// Mitsubishi GX Works2 project: 20250407_최종프로젝트_PLC_완성   PLC: Q03UDE

// global labels: Global1
VAR_GLOBAL
  압착1전솔 AT Y30 : BOOL;
  압착2전솔 AT Y31 : BOOL;
  배출전솔 AT Y32 : BOOL;
  회전전솔 AT Y34 : BOOL;
  회전후솔 AT Y35 : BOOL;
  스탑전솔 AT Y36 : BOOL;
  스탑후솔 AT Y37 : BOOL;
  서보전솔 AT Y38 : BOOL;
  서보후솔 AT Y39 : BOOL;
  컨베이어1 AT Y20 : BOOL;
  컨베이어2 AT Y21 : BOOL;
  컨베이어3 AT Y22 : BOOL;
  컨베이어4 AT Y23 : BOOL;
  스톱전센서 AT X1 : BOOL;
  스톱후센서 AT X0 : BOOL;
  스톱감지광센서 AT X2 : BOOL;
  두봇감지광센서1 AT X3 : BOOL;
  압착하강센서1 AT X5 : BOOL;
  회전상승센서 AT X7 : BOOL;
  회전하강센서 AT X8 : BOOL;
  배출감지광센서 AT X9 : BOOL;
  포장감지광센서1 AT X0A : BOOL;
  압착상승센서2 AT X0B : BOOL;
  압착하강센서2 AT X0C : BOOL;
  서보적재전센서 AT X0D : BOOL;
  서보적재후센서 AT X0E : BOOL;
  압착상승센서1 AT X6 : BOOL;
  포장감지광센서2 AT X10 : BOOL;
  회전감지광센서 AT X11 : BOOL;
  배출후센서 AT X13 : BOOL;
  배출전센서 AT X12 : BOOL;
  압착감지광센서 AT X14 : BOOL;
  두봇1빨강 AT Y2C : BOOL;
  두봇1하늘 AT Y2D : BOOL;
  두봇1노랑 AT Y2E : BOOL;
  두봇2동작1 AT Y2B : BOOL;
  축1서보기동번호 AT U4\G1500 : DINT;
  축1서보조그스피드값 AT U4\G1518 : DINT;
  축1서보현재위치 AT U4\G800 : DINT;
  축1서보이송속도 AT U4\G804 : DINT;
  축1서보원점복귀완료 AT U4\G817.4 : BOOL;
  QD75레디 AT X40 : BOOL;
  축1서보비지 AT X4C : BOOL;
  축1서보완료 AT X54 : BOOL;
  PLC레디 AT Y40 : BOOL;
  축1서보정지 AT Y44 : BOOL;
  축1서보조그정기동 AT Y48 : BOOL;
  축1서보조그역기동 AT Y49 : BOOL;
  축1서보기동 AT Y50 : BOOL;
  축2서보기동번호 AT U4\G1600 : DINT;
  축2서보조그스피드값 AT U4\G1618 : DINT;
  축2서보현재위치 AT U4\G900 : DINT;
  축2서보이송속도 AT U4\G904 : DINT;
  축2서보원점복귀완료 AT U4\G917.4 : BOOL;
  축2서보비지 AT X4B : BOOL;
  축2서보완료 AT X55 : BOOL;
  축2서보정지 AT Y45 : BOOL;
  축2서보조그정기동 AT Y4A : BOOL;
  축2서보조그역기동 AT Y4B : BOOL;
  축2서보기동 AT Y51 : BOOL;
  축1서보현재위치표시 AT D0 : DINT;
  축2서보현재위치표시 AT D10 : DINT;
  축1서보조그속도 AT D20 : DINT;
  축2서보조그속도 AT D30 : DINT;
  H1조그상 AT M0 : BOOL;
  H1조그하 AT M1 : BOOL;
  H2조그상 AT M2 : BOOL;
  H2조그하 AT M3 : BOOL;
  H1원점복귀버튼 AT M4 : BOOL;
  축1에러번호 AT U4\G806 : INT;
  축2에러번호 AT U4\G906 : INT;
  축1경고번호 AT U4\G807 : INT;
  축2경고번호 AT U4\G907 : INT;
  H시작버튼 AT M5 : BOOL;
  H일시정지버튼 AT M6 : BOOL;
  H비상정지버튼 AT M7 : BOOL;
  녹색램프 AT Y24 : BOOL;
  황색램프 AT Y25 : BOOL;
  적색램프 AT Y26 : BOOL;
  H축1원점복귀버튼 AT M8 : BOOL;
  H축2원점복귀버튼 AT M9 : BOOL;
  H롬저장 AT M200 : BOOL;
  서보롬쓰기 AT U4\G1900 : INT;
  H축1위치1입력 AT M300 : BOOL;
  H축1위치2입력 AT M301 : BOOL;
  H축1위치3입력 AT M302 : BOOL;
  H축2위치1입력 AT M310 : BOOL;
  H축2위치2입력 AT M311 : BOOL;
  H축2위치3입력 AT M312 : BOOL;
  H축2위치4입력 AT M313 : BOOL;
  H축2위치5입력 AT M314 : BOOL;
  H축2위치6입력 AT M315 : BOOL;
  H서보전진버튼 AT M10 : BOOL;
  H서보후진버튼 AT M11 : BOOL;
  H축1경고번호 AT D100 : INT;
  H축1에러번호 AT D101 : INT;
  H축2경고번호 AT D200 : INT;
  H축2에러번호 AT D201 : INT;
  H축1에러리셋 AT M400 : BOOL;
  H축2에러리셋 AT M401 : BOOL;
  축1에러리셋 AT U4\G1502 : INT;
  축2에러리셋 AT U4\G1602 : INT;
  송신채널 AT D1000 : INT;
  송신데이터수 AT D1002 : INT;
  송신데이터 AT D1010 : INT;
  수신채널 AT D1100 : INT;
  수신데이터수 AT D1103 : INT;
  수신버퍼 AT D1110 : INT;
  데이터체크 AT D1200 : INT;
  수신데이터확인 AT X6A : BOOL;
  송신정상 AT M1000 : BOOL;
  수신정상 AT M1100 : BOOL;
  두봇1완료 AT X18 : BOOL;
  두봇2완료 AT X19 : BOOL;
  H실린더스톱전진 AT M100 : BOOL;
  H실린더배출전진 AT M102 : BOOL;
  H실린더서보전진 AT M103 : BOOL;
  H실린더서보후진 AT M104 : BOOL;
  H실린더회전전진 AT M105 : BOOL;
  H실린더회전후진 AT M106 : BOOL;
  H실린더스톱후진 AT M101 : BOOL;
  H실린더압착전진1 AT M107 : BOOL;
  H실린더압착전진2 AT M108 : BOOL;
  H모터컨베이어1 AT M109 : BOOL;
  H모터컨베이어2 AT M110 : BOOL;
  H모터컨베이어3 AT M111 : BOOL;
  H모터컨베이어4 AT M112 : BOOL;
  S공정1_CT AT D3000 : INT;
  S공정2_CT AT D3002 : INT;
  S공정3_CT AT D3004 : INT;
  S공정4_CT AT D3006 : INT;
  축1서보조그속도표시 AT D40 : DINT;
  축2서보조그속도표시 AT D50 : DINT;
  S양품갯수 AT D3008 : INT;
  S불량갯수 AT D3010 : INT;
  S적재갯수 AT D3012 : INT;
  S고배율갯수 AT D3014 : INT;
  S중배율갯수 AT D3015 : INT;
  S저배율갯수 AT D3016 : INT;
  S고배율 AT D3017 : INT;
  S중배율 AT D3018 : INT;
  S저배율 AT D3019 : INT;
  두봇2동작중 AT M17 : BOOL;
  두봇1동작중 AT M16 : BOOL;
  녹색램프버튼 AT M30 : BOOL;
  황색램프버튼 AT M31 : BOOL;
  적색램프버튼 AT M32 : BOOL;
END_VAR

PROGRAM MAIN
VAR
  공정시작 : BOOL;
  축2기동 : BOOL;
  축1기동 : BOOL;
  공정종료 : BOOL;
  스톱후진 : BOOL;
  컨베이어1구동 : BOOL;
  컨베이어1정지 : BOOL;
  스톱전진 : BOOL;
  T스톱지연 : TIMER;
  서보준비완료 : BOOL;
  두봇앞정지 : BOOL;
  컨베이어1정지2 : BOOL;
  T두봇지연 : TIMER;
  압착앞이동 : BOOL;
  압착압이동 : BOOL;
  압착1전진 : BOOL;
  압착1후진 : BOOL;
  컨베이어1정지3 : BOOL;
  압착전진 : BOOL;
  압착후진 : BOOL;
  컨베이어1종료 : BOOL;
  T컨베이어1지연 : TIMER;
  컨베이어2구동 : BOOL;
  공정1종료 : BOOL;
  컨베이어1정지4 : BOOL;
  컨베이어4구동 : BOOL;
  T불량품감지 : TIMER;
  컨베이어3구동 : BOOL;
  컨베이어2정지1 : BOOL;
  비전감지 : BOOL;
  T비전감지지연 : TIMER;
  양품판별 : BOOL;
  불량판별 : BOOL;
  T두봇지연2 : TIMER;
  T포장1지연 : TIMER;
  T두봇지연3 : TIMER;
  T압착지연 : TIMER;
  압착2전진 : BOOL;
  압착2후진 : BOOL;
  회전전진 : BOOL;
  서보위치1이동 : BOOL;
  서보전진 : BOOL;
  T회전지연 : TIMER;
  T비상정지초기화 : TIMER;
  포장대기 : BOOL;
  포장대기2 : BOOL;
  축1위치1이동 : BOOL;
  축2위치1이동 : BOOL;
  T서보전진지연 : TIMER;
  서보후진 : BOOL;
  T서보후진지연 : TIMER;
  축2위치2이동 : BOOL;
  회전후진 : BOOL;
  축2위치3이동 : BOOL;
  축1위치2이동 : BOOL;
  축2위치4이동 : BOOL;
  T서보전진지연2 : TIMER;
  축1위치1이동2 : BOOL;
  축2위치1이동2 : BOOL;
  축2위치3이동2 : BOOL;
  회전대기 : BOOL;
  축1원점복귀 : BOOL;
  축2원점복귀 : BOOL;
  양품개수 : INT;
  연속종료 : BOOL;
  서보적재후진 : BOOL;
  롬쓰기 : BOOL;
  H롬쓰기 : BOOL;
  축1조그스피드값 : DINT;
  축2조그스피드값 : DINT;
  T압착정지지연 : TIMER;
  T압착정지지연2 : TIMER;
  공정중 : BOOL;
  적재완료대기 : BOOL;
  스톱후진2 : BOOL;
  T회전후진지연 : TIMER;
  시작 : BOOL;
  종료복귀 : BOOL;
  축1복귀1이동 : BOOL;
  복귀종료 : BOOL;
  축2복귀1이동 : BOOL;
  축1복귀2이동 : BOOL;
  종료 : BOOL;
  T불량판별지연 : TIMER;
  배출전진 : BOOL;
  배출후진 : BOOL;
  불량종료 : BOOL;
  양품종료 : BOOL;
  컨종료 : BOOL;
  T컨종료지연 : TIMER;
  두봇사양구별 : BOOL;
  두봇1완료신호 : BOOL;
  T포장대기지연 : TIMER;
  두봇포장완료 : BOOL;
  T컨베이어4지연 : TIMER;
  테스트 : BOOL;
  공정1그래프 : BOOL;
  공정2그래프 : BOOL;
  공정3그래프 : BOOL;
  공정4그래프 : BOOL;
  공정1CT : INT;
  공정2CT : INT;
  공정3CT : INT;
  공정4CT : INT;
  불량개수 : INT;
  적재완료 : BOOL;
  스톱후진3 : BOOL;
  두봇2동작 : BOOL;
  축1일시정지요구 : BOOL;
  축2일시정지요구 : BOOL;
  축2비상정지요구 : BOOL;
  축1비상정지요구 : BOOL;
  비상정지요구 : BOOL;
  일시정지요구 : BOOL;
  T축2일시정지기동 : TIMER;
  일시정지풀림 : BOOL;
END_VAR
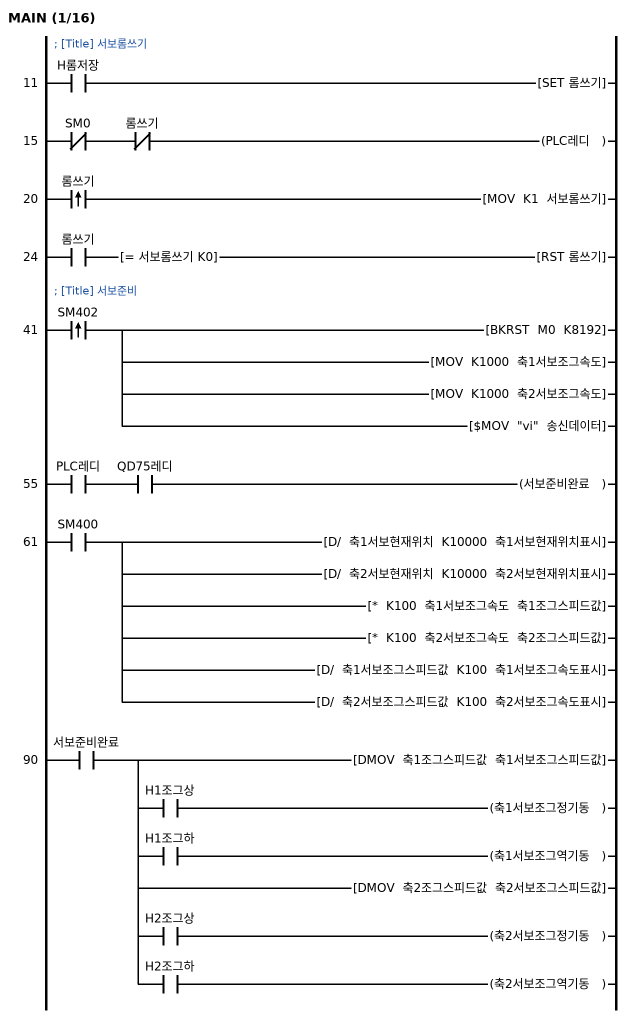
; [Title] 서보롬쓰기
11    LD      H롬저장
      SET     롬쓰기
15    LDI     SM0
      ANI     롬쓰기
      OUT     PLC레디
20    LDP     롬쓰기
      MOV     K1 서보롬쓰기
24    LD      롬쓰기
      AND=    서보롬쓰기 K0
      RST     롬쓰기
; [Title] 서보준비
41    LDP     SM402
      BKRST   M0 K8192
      MOV     K1000 축1서보조그속도
      MOV     K1000 축2서보조그속도
      $MOV    "vi" 송신데이터
55    LD      PLC레디
      AND     QD75레디
      OUT     서보준비완료
61    LD      SM400
      D/      축1서보현재위치 K10000 축1서보현재위치표시
      D/      축2서보현재위치 K10000 축2서보현재위치표시
      *       K100 축1서보조그속도 축1조그스피드값
      *       K100 축2서보조그속도 축2조그스피드값
      D/      축1서보조그스피드값 K100 축1서보조그속도표시
      D/      축2서보조그스피드값 K100 축2서보조그속도표시
90    LD      서보준비완료
      DMOV    축1조그스피드값 축1서보조그스피드값
      MPS
      AND     H1조그상
      OUT     축1서보조그정기동
      MRD
      AND     H1조그하
      OUT     축1서보조그역기동
      MPP
      DMOV    축2조그스피드값 축2서보조그스피드값
      MPS
      AND     H2조그상
      OUT     축2서보조그정기동
      MPP
      AND     H2조그하
      OUT     축2서보조그역기동
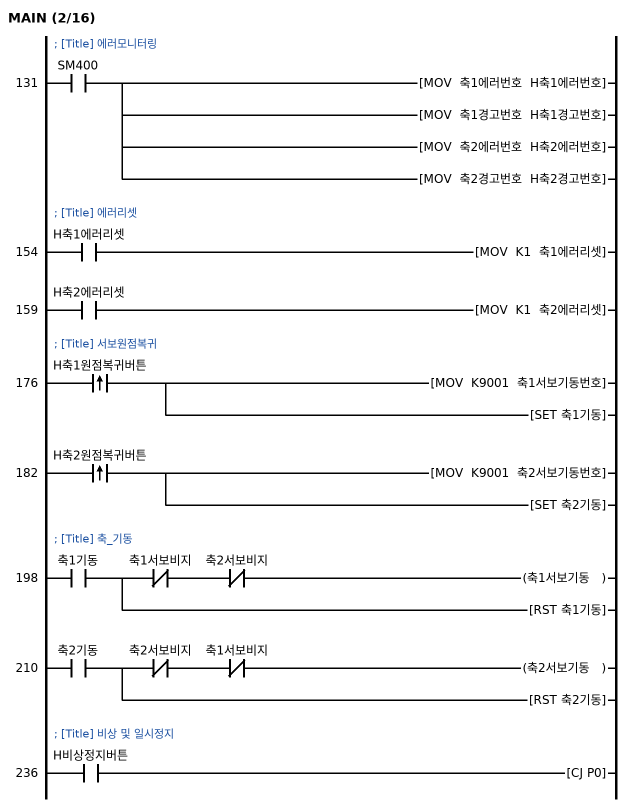
; [Title] 에러모니터링
131   LD      SM400
      MOV     축1에러번호 H축1에러번호
      MOV     축1경고번호 H축1경고번호
      MOV     축2에러번호 H축2에러번호
      MOV     축2경고번호 H축2경고번호
; [Title] 에러리셋
154   LD      H축1에러리셋
      MOV     K1 축1에러리셋
159   LD      H축2에러리셋
      MOV     K1 축2에러리셋
; [Title] 서보원점복귀
176   LDP     H축1원점복귀버튼
      MOV     K9001 축1서보기동번호
      SET     축1기동
182   LDP     H축2원점복귀버튼
      MOV     K9001 축2서보기동번호
      SET     축2기동
; [Title] 축_기동
198   LD      축1기동
      MPS
      ANI     축1서보비지
      ANI     축2서보비지
      OUT     축1서보기동
      MPP
      RST     축1기동
210   LD      축2기동
      MPS
      ANI     축2서보비지
      ANI     축1서보비지
      OUT     축2서보기동
      MPP
      RST     축2기동
; [Title] 비상 및 일시정지
236   LD      H비상정지버튼
      CJ      P0
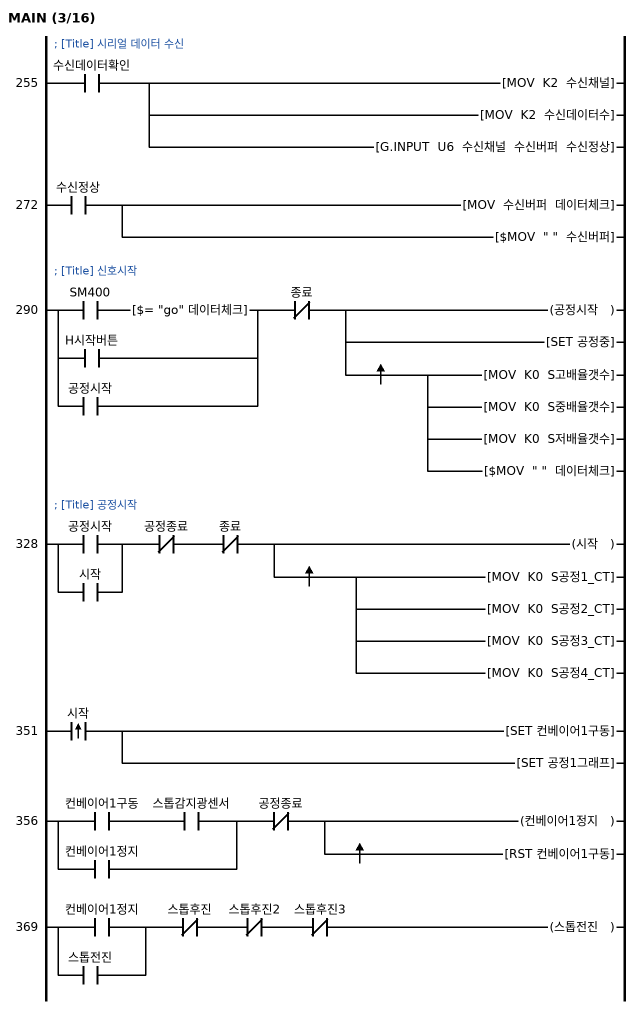
; [Title] 시리얼 데이터 수신
255   LD      수신데이터확인
      MOV     K2 수신채널
      MOV     K2 수신데이터수
      G.INPUT U6 수신채널 수신버퍼 수신정상
272   LD      수신정상
      MOV     수신버퍼 데이터체크
      $MOV    "" 수신버퍼
; [Title] 신호시작
290   LD      SM400
      AND$=   "go" 데이터체크
      OR      H시작버튼
      OR      공정시작
      ANI     종료
      OUT     공정시작
      SET     공정중
      MEP
      MOV     K0 S고배율갯수
      MOV     K0 S중배율갯수
      MOV     K0 S저배율갯수
      $MOV    "" 데이터체크
; [Title] 공정시작
328   LD      공정시작
      OR      시작
      ANI     공정종료
      ANI     종료
      OUT     시작
      MEP
      MOV     K0 S공정1_CT
      MOV     K0 S공정2_CT
      MOV     K0 S공정3_CT
      MOV     K0 S공정4_CT
351   LDP     시작
      SET     컨베이어1구동
      SET     공정1그래프
356   LD      컨베이어1구동
      AND     스톱감지광센서
      OR      컨베이어1정지
      ANI     공정종료
      OUT     컨베이어1정지
      MEP
      RST     컨베이어1구동
369   LD      컨베이어1정지
      OR      스톱전진
      ANI     스톱후진
      ANI     스톱후진2
      ANI     스톱후진3
      OUT     스톱전진
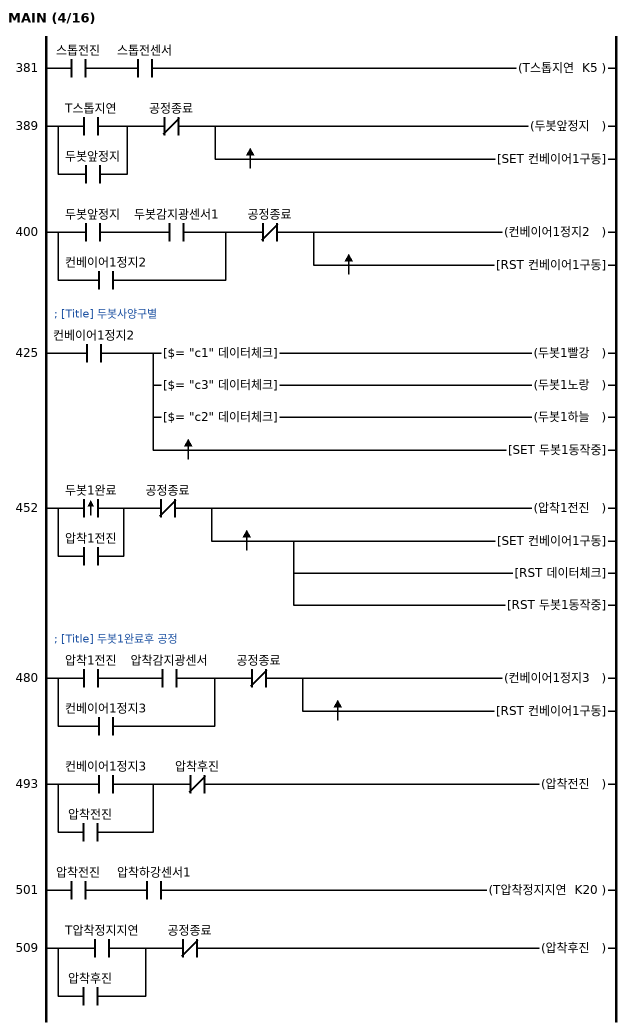
381   LD      스톱전진
      AND     스톱전센서
      OUT     T스톱지연 K5
389   LD      T스톱지연
      OR      두봇앞정지
      ANI     공정종료
      OUT     두봇앞정지
      MEP
      SET     컨베이어1구동
400   LD      두봇앞정지
      AND     두봇감지광센서1
      OR      컨베이어1정지2
      ANI     공정종료
      OUT     컨베이어1정지2
      MEP
      RST     컨베이어1구동
; [Title] 두봇사양구별
425   LD      컨베이어1정지2
      MPS
      AND$=   "c1" 데이터체크
      OUT     두봇1빨강
      MRD
      AND$=   "c3" 데이터체크
      OUT     두봇1노랑
      MRD
      AND$=   "c2" 데이터체크
      OUT     두봇1하늘
      MPP
      MEP
      SET     두봇1동작중
452   LDP     두봇1완료
      OR      압착1전진
      ANI     공정종료
      OUT     압착1전진
      MEP
      SET     컨베이어1구동
      RST     데이터체크
      RST     두봇1동작중
; [Title] 두봇1완료후 공정
480   LD      압착1전진
      AND     압착감지광센서
      OR      컨베이어1정지3
      ANI     공정종료
      OUT     컨베이어1정지3
      MEP
      RST     컨베이어1구동
493   LD      컨베이어1정지3
      OR      압착전진
      ANI     압착후진
      OUT     압착전진
501   LD      압착전진
      AND     압착하강센서1
      OUT     T압착정지지연 K20
509   LD      T압착정지지연
      OR      압착후진
      ANI     공정종료
      OUT     압착후진
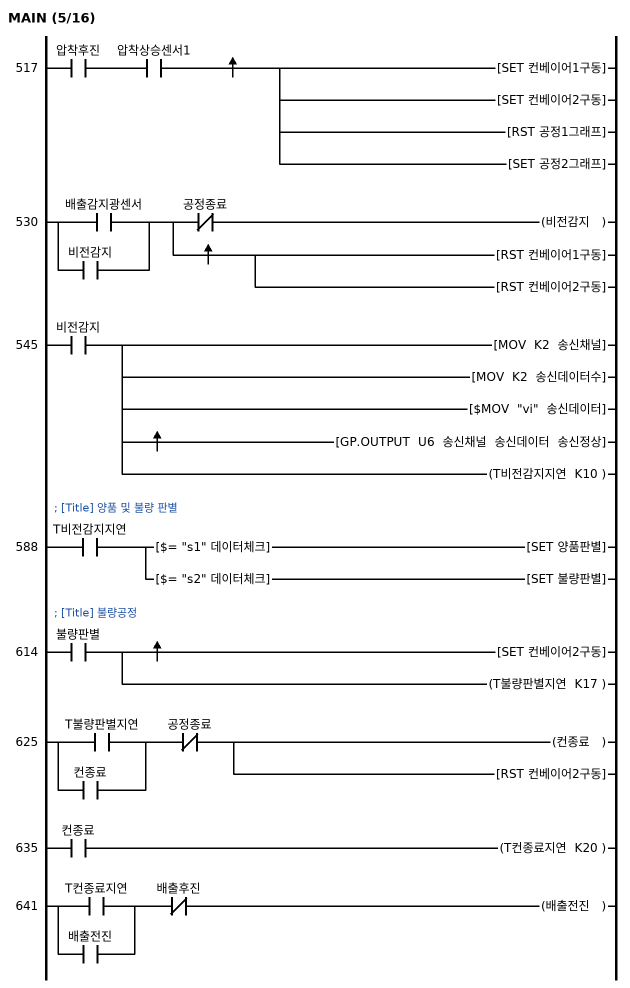
517   LD      압착후진
      AND     압착상승센서1
      MEP
      SET     컨베이어1구동
      SET     컨베이어2구동
      RST     공정1그래프
      SET     공정2그래프
530   LD      배출감지광센서
      OR      비전감지
      MPS
      ANI     공정종료
      OUT     비전감지
      MPP
      MEP
      RST     컨베이어1구동
      RST     컨베이어2구동
545   LD      비전감지
      MOV     K2 송신채널
      MOV     K2 송신데이터수
      $MOV    "vi" 송신데이터
      MPS
      MEP
      GP.OUTPUT U6 송신채널 송신데이터 송신정상
      MPP
      OUT     T비전감지지연 K10
; [Title] 양품 및 불량 판별
588   LD      T비전감지지연
      MPS
      AND$=   "s1" 데이터체크
      SET     양품판별
      MPP
      AND$=   "s2" 데이터체크
      SET     불량판별
; [Title] 불량공정
614   LD      불량판별
      MPS
      MEP
      SET     컨베이어2구동
      MPP
      OUT     T불량판별지연 K17
625   LD      T불량판별지연
      OR      컨종료
      ANI     공정종료
      OUT     컨종료
      RST     컨베이어2구동
635   LD      컨종료
      OUT     T컨종료지연 K20
641   LD      T컨종료지연
      OR      배출전진
      ANI     배출후진
      OUT     배출전진
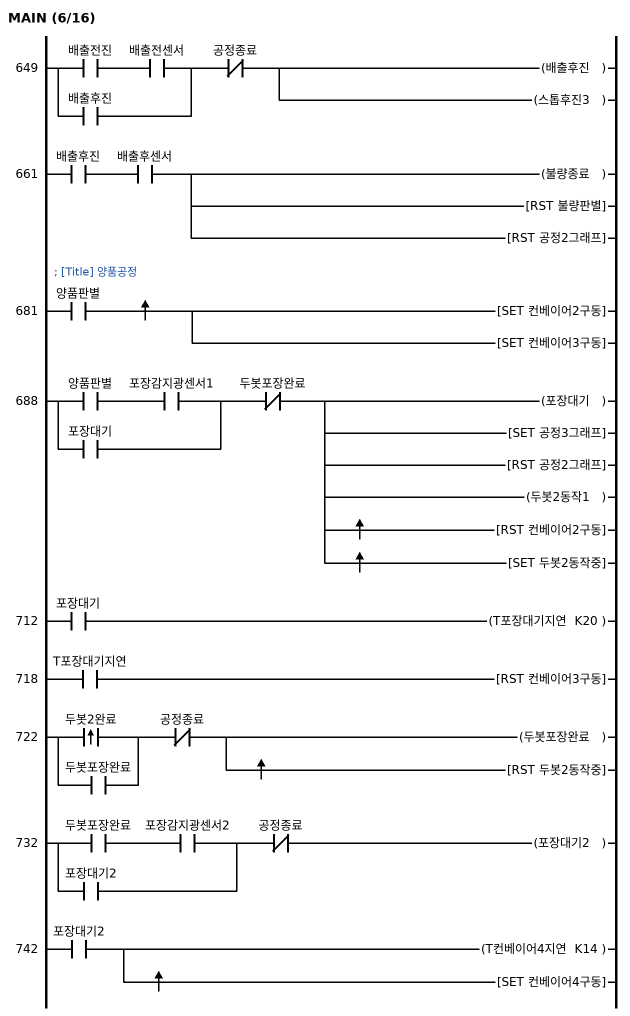
649   LD      배출전진
      AND     배출전센서
      OR      배출후진
      ANI     공정종료
      OUT     배출후진
      OUT     스톱후진3
661   LD      배출후진
      AND     배출후센서
      OUT     불량종료
      RST     불량판별
      RST     공정2그래프
; [Title] 양품공정
681   LD      양품판별
      MEP
      SET     컨베이어2구동
      SET     컨베이어3구동
688   LD      양품판별
      AND     포장감지광센서1
      OR      포장대기
      ANI     두봇포장완료
      OUT     포장대기
      SET     공정3그래프
      RST     공정2그래프
      OUT     두봇2동작1
      MPS
      MEP
      RST     컨베이어2구동
      MPP
      MEP
      SET     두봇2동작중
712   LD      포장대기
      OUT     T포장대기지연 K20
718   LD      T포장대기지연
      RST     컨베이어3구동
722   LDP     두봇2완료
      OR      두봇포장완료
      ANI     공정종료
      OUT     두봇포장완료
      MEP
      RST     두봇2동작중
732   LD      두봇포장완료
      AND     포장감지광센서2
      OR      포장대기2
      ANI     공정종료
      OUT     포장대기2
742   LD      포장대기2
      OUT     T컨베이어4지연 K14
      MEP
      SET     컨베이어4구동
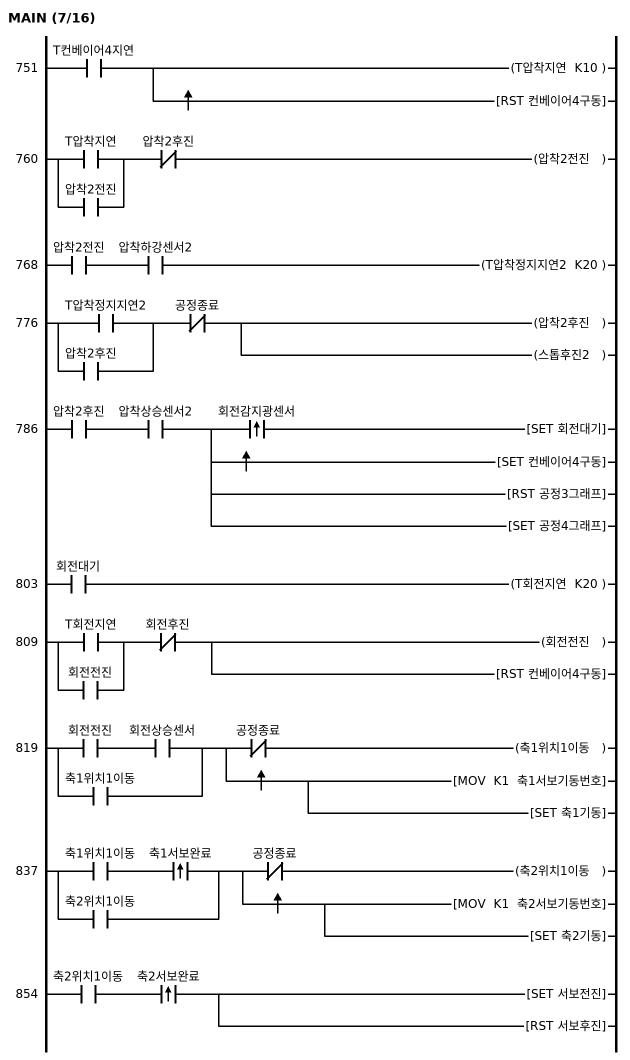
751   LD      T컨베이어4지연
      OUT     T압착지연 K10
      MEP
      RST     컨베이어4구동
760   LD      T압착지연
      OR      압착2전진
      ANI     압착2후진
      OUT     압착2전진
768   LD      압착2전진
      AND     압착하강센서2
      OUT     T압착정지지연2 K20
776   LD      T압착정지지연2
      OR      압착2후진
      ANI     공정종료
      OUT     압착2후진
      OUT     스톱후진2
786   LD      압착2후진
      AND     압착상승센서2
      MPS
      ANDP    회전감지광센서
      SET     회전대기
      MRD
      MEP
      SET     컨베이어4구동
      MPP
      RST     공정3그래프
      SET     공정4그래프
803   LD      회전대기
      OUT     T회전지연 K20
809   LD      T회전지연
      OR      회전전진
      ANI     회전후진
      OUT     회전전진
      RST     컨베이어4구동
819   LD      회전전진
      AND     회전상승센서
      OR      축1위치1이동
      MPS
      ANI     공정종료
      OUT     축1위치1이동
      MPP
      MEP
      MOV     K1 축1서보기동번호
      SET     축1기동
837   LD      축1위치1이동
      ANDP    축1서보완료
      OR      축2위치1이동
      MPS
      ANI     공정종료
      OUT     축2위치1이동
      MPP
      MEP
      MOV     K1 축2서보기동번호
      SET     축2기동
854   LD      축2위치1이동
      ANDP    축2서보완료
      SET     서보전진
      RST     서보후진
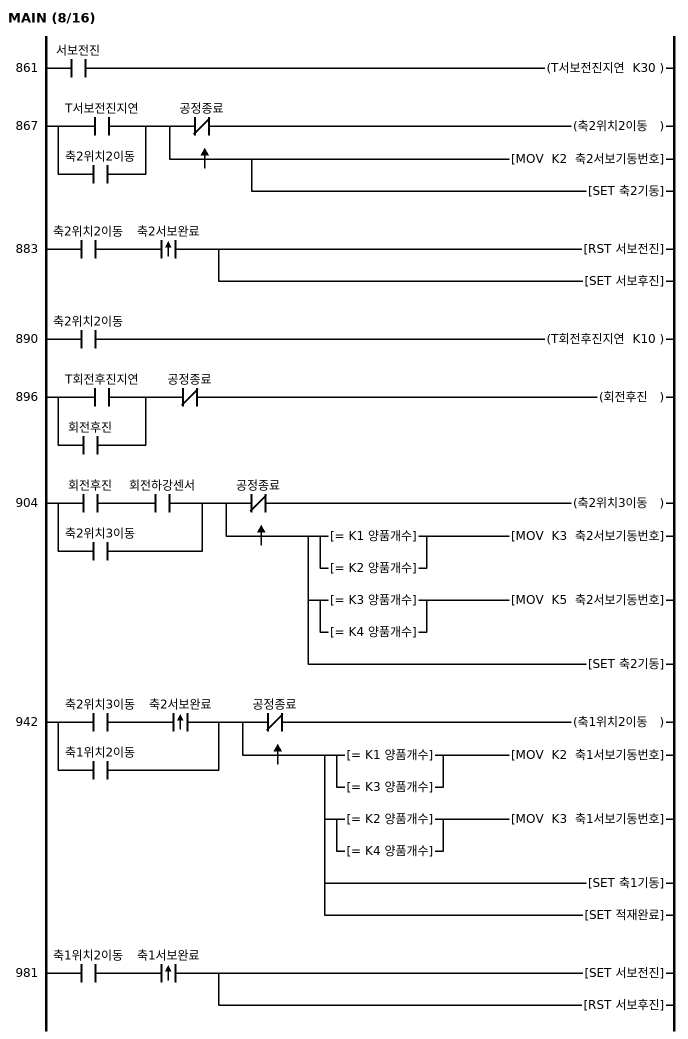
861   LD      서보전진
      OUT     T서보전진지연 K30
867   LD      T서보전진지연
      OR      축2위치2이동
      MPS
      ANI     공정종료
      OUT     축2위치2이동
      MPP
      MEP
      MOV     K2 축2서보기동번호
      SET     축2기동
883   LD      축2위치2이동
      ANDP    축2서보완료
      RST     서보전진
      SET     서보후진
890   LD      축2위치2이동
      OUT     T회전후진지연 K10
896   LD      T회전후진지연
      OR      회전후진
      ANI     공정종료
      OUT     회전후진
904   LD      회전후진
      AND     회전하강센서
      OR      축2위치3이동
      MPS
      ANI     공정종료
      OUT     축2위치3이동
      MPP
      MEP
      MPS
      LD=     K1 양품개수
      OR=     K2 양품개수
      ANB
      MOV     K3 축2서보기동번호
      MRD
      LD=     K3 양품개수
      OR=     K4 양품개수
      ANB
      MOV     K5 축2서보기동번호
      MPP
      SET     축2기동
942   LD      축2위치3이동
      ANDP    축2서보완료
      OR      축1위치2이동
      MPS
      ANI     공정종료
      OUT     축1위치2이동
      MPP
      MEP
      MPS
      LD=     K1 양품개수
      OR=     K3 양품개수
      ANB
      MOV     K2 축1서보기동번호
      MRD
      LD=     K2 양품개수
      OR=     K4 양품개수
      ANB
      MOV     K3 축1서보기동번호
      MPP
      SET     축1기동
      SET     적재완료
981   LD      축1위치2이동
      ANDP    축1서보완료
      SET     서보전진
      RST     서보후진
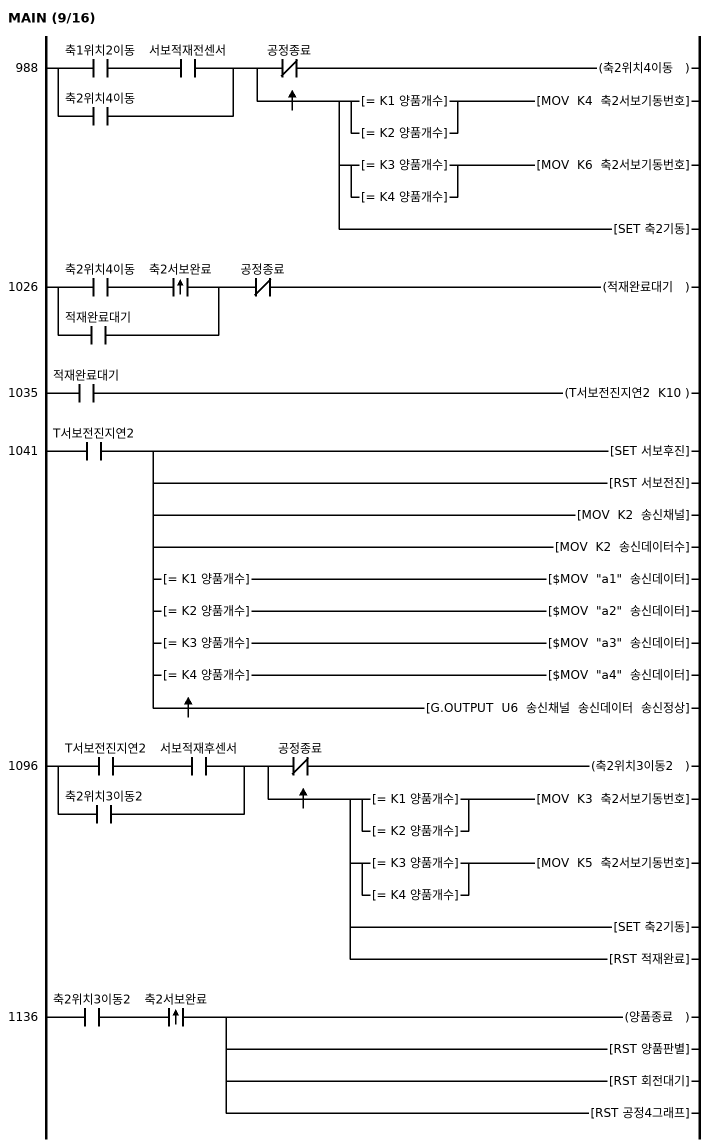
988   LD      축1위치2이동
      AND     서보적재전센서
      OR      축2위치4이동
      MPS
      ANI     공정종료
      OUT     축2위치4이동
      MPP
      MEP
      MPS
      LD=     K1 양품개수
      OR=     K2 양품개수
      ANB
      MOV     K4 축2서보기동번호
      MRD
      LD=     K3 양품개수
      OR=     K4 양품개수
      ANB
      MOV     K6 축2서보기동번호
      MPP
      SET     축2기동
1026  LD      축2위치4이동
      ANDP    축2서보완료
      OR      적재완료대기
      ANI     공정종료
      OUT     적재완료대기
1035  LD      적재완료대기
      OUT     T서보전진지연2 K10
1041  LD      T서보전진지연2
      SET     서보후진
      RST     서보전진
      MOV     K2 송신채널
      MOV     K2 송신데이터수
      MPS
      AND=    K1 양품개수
      $MOV    "a1" 송신데이터
      MRD
      AND=    K2 양품개수
      $MOV    "a2" 송신데이터
      MRD
      AND=    K3 양품개수
      $MOV    "a3" 송신데이터
      MRD
      AND=    K4 양품개수
      $MOV    "a4" 송신데이터
      MPP
      MEP
      G.OUTPUT U6 송신채널 송신데이터 송신정상
1096  LD      T서보전진지연2
      AND     서보적재후센서
      OR      축2위치3이동2
      MPS
      ANI     공정종료
      OUT     축2위치3이동2
      MPP
      MEP
      MPS
      LD=     K1 양품개수
      OR=     K2 양품개수
      ANB
      MOV     K3 축2서보기동번호
      MRD
      LD=     K3 양품개수
      OR=     K4 양품개수
      ANB
      MOV     K5 축2서보기동번호
      MPP
      SET     축2기동
      RST     적재완료
1136  LD      축2위치3이동2
      ANDP    축2서보완료
      OUT     양품종료
      RST     양품판별
      RST     회전대기
      RST     공정4그래프
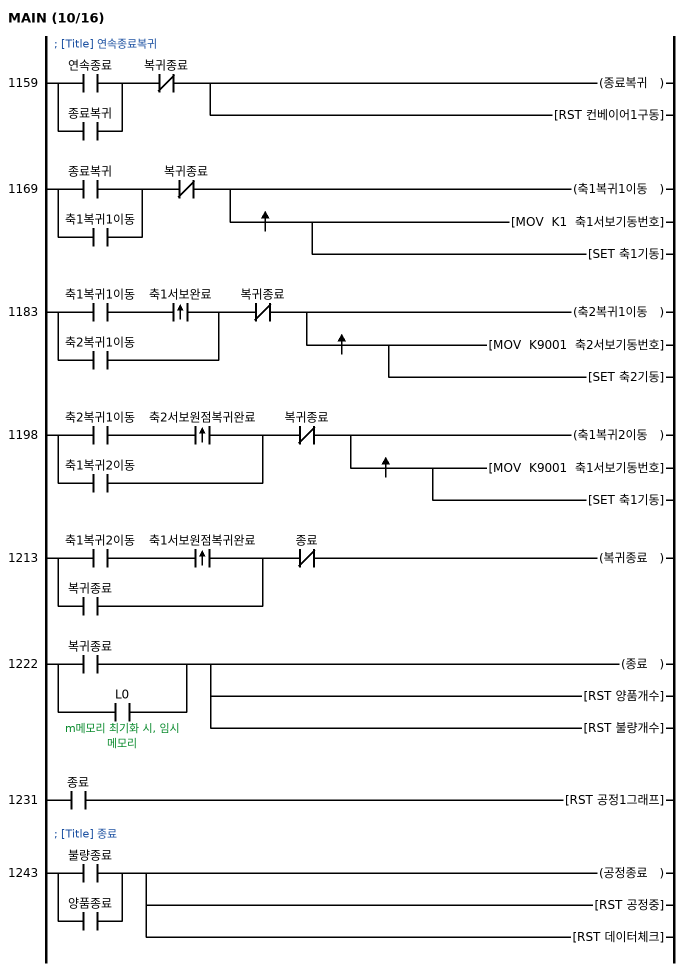
; [Title] 연속종료복귀
1159  LD      연속종료
      OR      종료복귀
      ANI     복귀종료
      OUT     종료복귀
      RST     컨베이어1구동
1169  LD      종료복귀
      OR      축1복귀1이동
      ANI     복귀종료
      OUT     축1복귀1이동
      MEP
      MOV     K1 축1서보기동번호
      SET     축1기동
1183  LD      축1복귀1이동
      ANDP    축1서보완료
      OR      축2복귀1이동
      ANI     복귀종료
      OUT     축2복귀1이동
      MEP
      MOV     K9001 축2서보기동번호
      SET     축2기동
1198  LD      축2복귀1이동
      ANDP    축2서보원점복귀완료
      OR      축1복귀2이동
      ANI     복귀종료
      OUT     축1복귀2이동
      MEP
      MOV     K9001 축1서보기동번호
      SET     축1기동
1213  LD      축1복귀2이동
      ANDP    축1서보원점복귀완료
      OR      복귀종료
      ANI     종료
      OUT     복귀종료
1222  LD      복귀종료
      OR      L0  ; m메모리 최기화 시, 임시 메모리
      OUT     종료
      RST     양품개수
      RST     불량개수
1231  LD      종료
      RST     공정1그래프
; [Title] 종료
1243  LD      불량종료
      OR      양품종료
      OUT     공정종료
      RST     공정중
      RST     데이터체크
; [Title] 출력부
      P0
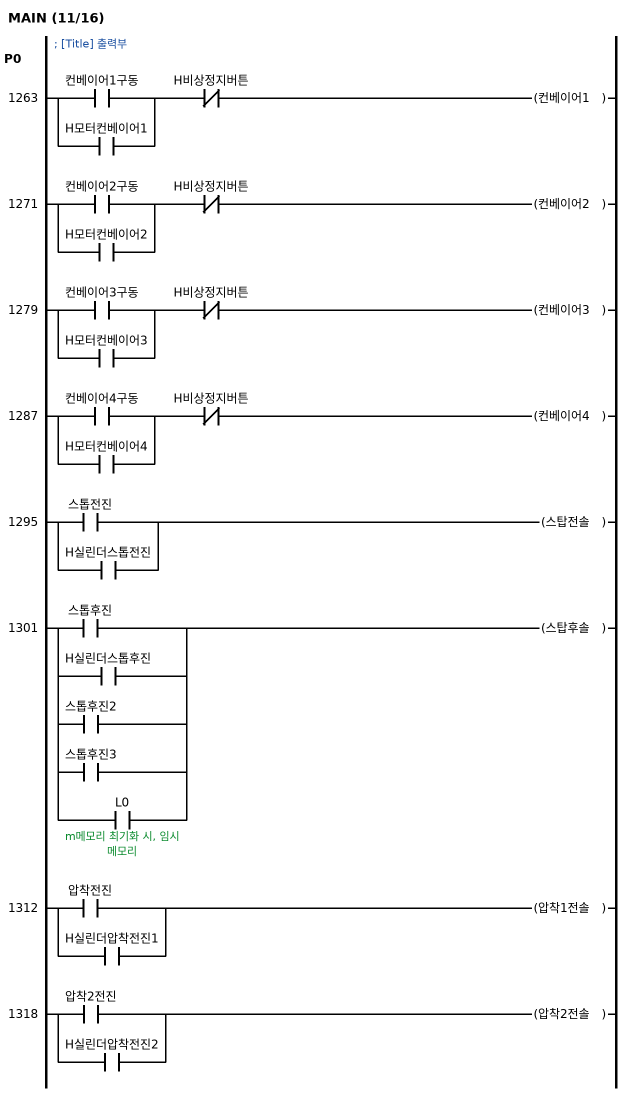
1263  LD      컨베이어1구동
      OR      H모터컨베이어1
      ANI     H비상정지버튼
      OUT     컨베이어1
1271  LD      컨베이어2구동
      OR      H모터컨베이어2
      ANI     H비상정지버튼
      OUT     컨베이어2
1279  LD      컨베이어3구동
      OR      H모터컨베이어3
      ANI     H비상정지버튼
      OUT     컨베이어3
1287  LD      컨베이어4구동
      OR      H모터컨베이어4
      ANI     H비상정지버튼
      OUT     컨베이어4
1295  LD      스톱전진
      OR      H실린더스톱전진
      OUT     스탑전솔
1301  LD      스톱후진
      OR      H실린더스톱후진
      OR      스톱후진2
      OR      스톱후진3
      OR      L0  ; m메모리 최기화 시, 임시 메모리
      OUT     스탑후솔
1312  LD      압착전진
      OR      H실린더압착전진1
      OUT     압착1전솔
1318  LD      압착2전진
      OR      H실린더압착전진2
      OUT     압착2전솔
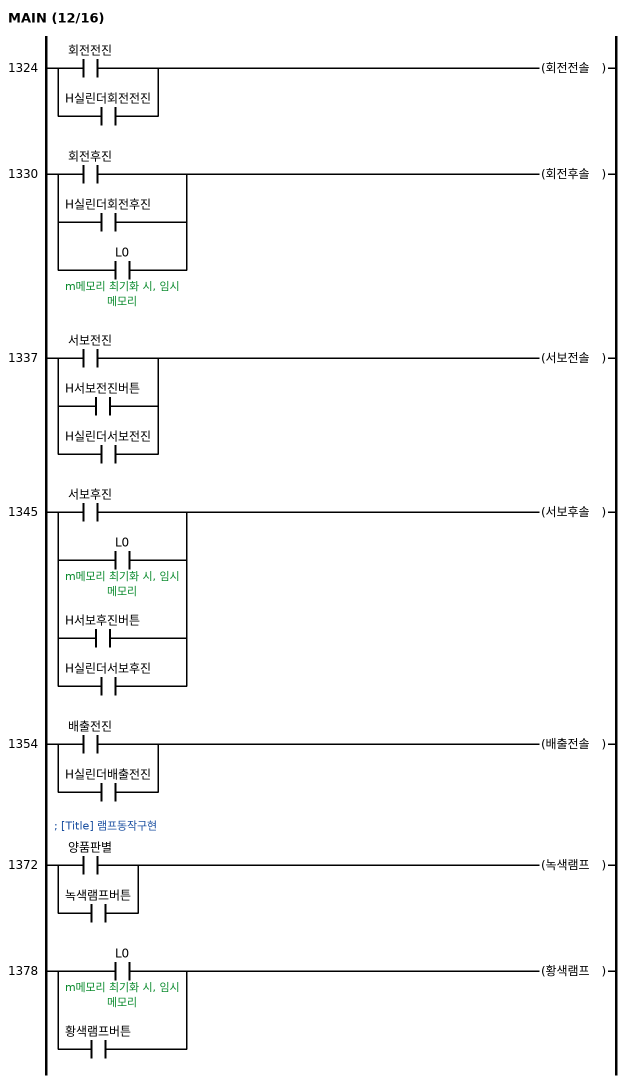
1324  LD      회전전진
      OR      H실린더회전전진
      OUT     회전전솔
1330  LD      회전후진
      OR      H실린더회전후진
      OR      L0  ; m메모리 최기화 시, 임시 메모리
      OUT     회전후솔
1337  LD      서보전진
      OR      H서보전진버튼
      OR      H실린더서보전진
      OUT     서보전솔
1345  LD      서보후진
      OR      L0  ; m메모리 최기화 시, 임시 메모리
      OR      H서보후진버튼
      OR      H실린더서보후진
      OUT     서보후솔
1354  LD      배출전진
      OR      H실린더배출전진
      OUT     배출전솔
; [Title] 램프동작구현
1372  LD      양품판별
      OR      녹색램프버튼
      OUT     녹색램프
1378  LD      L0  ; m메모리 최기화 시, 임시 메모리
      OR      황색램프버튼
      OUT     황색램프
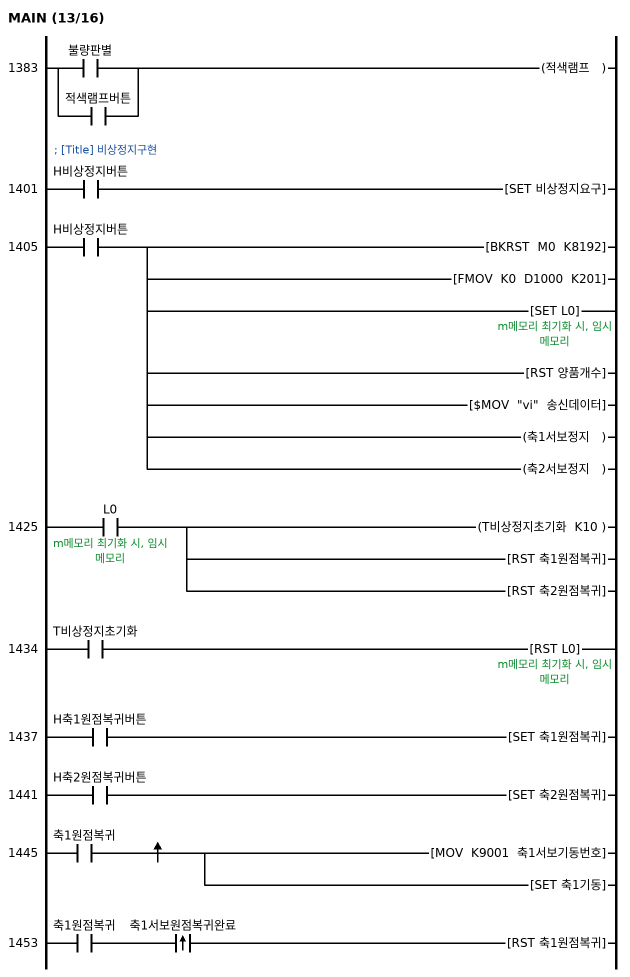
1383  LD      불량판별
      OR      적색램프버튼
      OUT     적색램프
; [Title] 비상정지구현
1401  LD      H비상정지버튼
      SET     비상정지요구
1405  LD      H비상정지버튼
      BKRST   M0 K8192
      FMOV    K0 D1000 K201
      SET     L0  ; m메모리 최기화 시, 임시 메모리
      RST     양품개수
      $MOV    "vi" 송신데이터
      OUT     축1서보정지
      OUT     축2서보정지
1425  LD      L0  ; m메모리 최기화 시, 임시 메모리
      OUT     T비상정지초기화 K10
      RST     축1원점복귀
      RST     축2원점복귀
1434  LD      T비상정지초기화
      RST     L0  ; m메모리 최기화 시, 임시 메모리
1437  LD      H축1원점복귀버튼
      SET     축1원점복귀
1441  LD      H축2원점복귀버튼
      SET     축2원점복귀
1445  LD      축1원점복귀
      MEP
      MOV     K9001 축1서보기동번호
      SET     축1기동
1453  LD      축1원점복귀
      ANDP    축1서보원점복귀완료
      RST     축1원점복귀
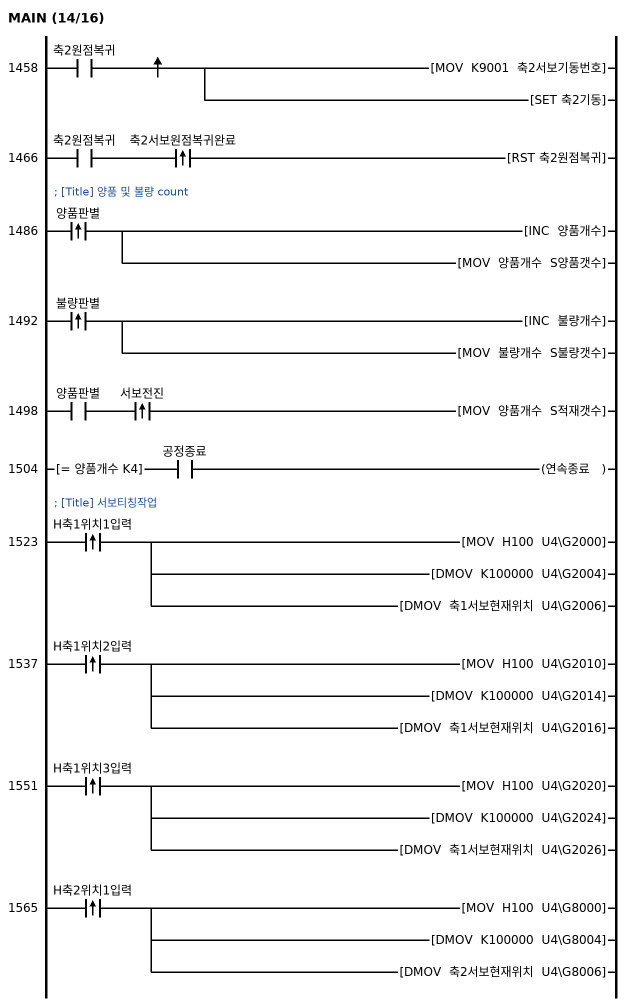
1458  LD      축2원점복귀
      MEP
      MOV     K9001 축2서보기동번호
      SET     축2기동
1466  LD      축2원점복귀
      ANDP    축2서보원점복귀완료
      RST     축2원점복귀
; [Title] 양품 및 불량 count
1486  LDP     양품판별
      INC     양품개수
      MOV     양품개수 S양품갯수
1492  LDP     불량판별
      INC     불량개수
      MOV     불량개수 S불량갯수
1498  LD      양품판별
      ANDP    서보전진
      MOV     양품개수 S적재갯수
1504  LD=     양품개수 K4
      AND     공정종료
      OUT     연속종료
; [Title] 서보티칭작업
1523  LDP     H축1위치1입력
      MOV     H100 U4\G2000
      DMOV    K100000 U4\G2004
      DMOV    축1서보현재위치 U4\G2006
1537  LDP     H축1위치2입력
      MOV     H100 U4\G2010
      DMOV    K100000 U4\G2014
      DMOV    축1서보현재위치 U4\G2016
1551  LDP     H축1위치3입력
      MOV     H100 U4\G2020
      DMOV    K100000 U4\G2024
      DMOV    축1서보현재위치 U4\G2026
1565  LDP     H축2위치1입력
      MOV     H100 U4\G8000
      DMOV    K100000 U4\G8004
      DMOV    축2서보현재위치 U4\G8006
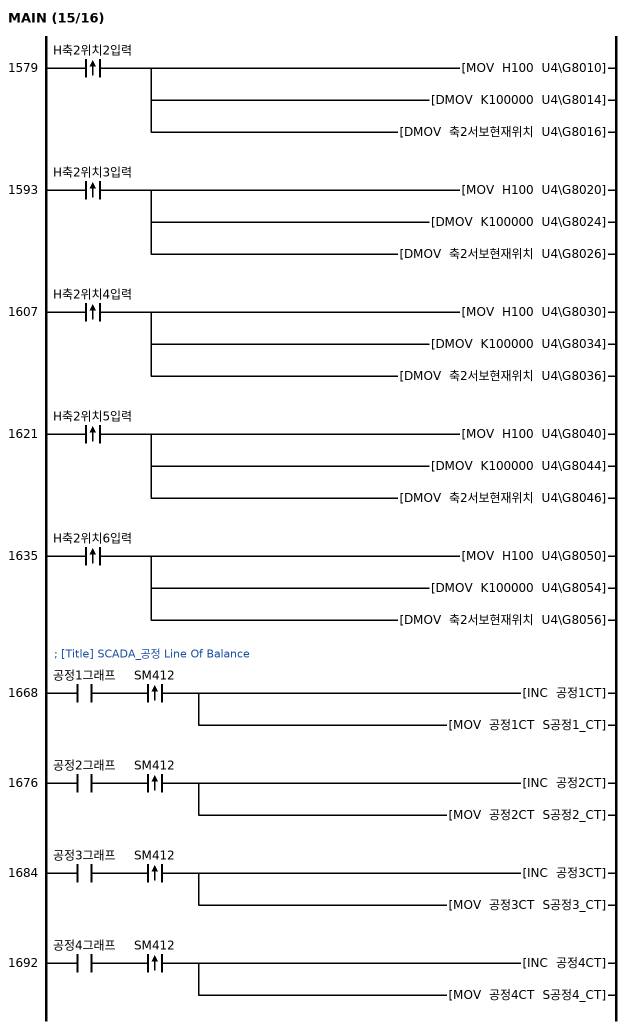
1579  LDP     H축2위치2입력
      MOV     H100 U4\G8010
      DMOV    K100000 U4\G8014
      DMOV    축2서보현재위치 U4\G8016
1593  LDP     H축2위치3입력
      MOV     H100 U4\G8020
      DMOV    K100000 U4\G8024
      DMOV    축2서보현재위치 U4\G8026
1607  LDP     H축2위치4입력
      MOV     H100 U4\G8030
      DMOV    K100000 U4\G8034
      DMOV    축2서보현재위치 U4\G8036
1621  LDP     H축2위치5입력
      MOV     H100 U4\G8040
      DMOV    K100000 U4\G8044
      DMOV    축2서보현재위치 U4\G8046
1635  LDP     H축2위치6입력
      MOV     H100 U4\G8050
      DMOV    K100000 U4\G8054
      DMOV    축2서보현재위치 U4\G8056
; [Title] SCADA_공정 Line Of Balance
1668  LD      공정1그래프
      ANDP    SM412
      INC     공정1CT
      MOV     공정1CT S공정1_CT
1676  LD      공정2그래프
      ANDP    SM412
      INC     공정2CT
      MOV     공정2CT S공정2_CT
1684  LD      공정3그래프
      ANDP    SM412
      INC     공정3CT
      MOV     공정3CT S공정3_CT
1692  LD      공정4그래프
      ANDP    SM412
      INC     공정4CT
      MOV     공정4CT S공정4_CT
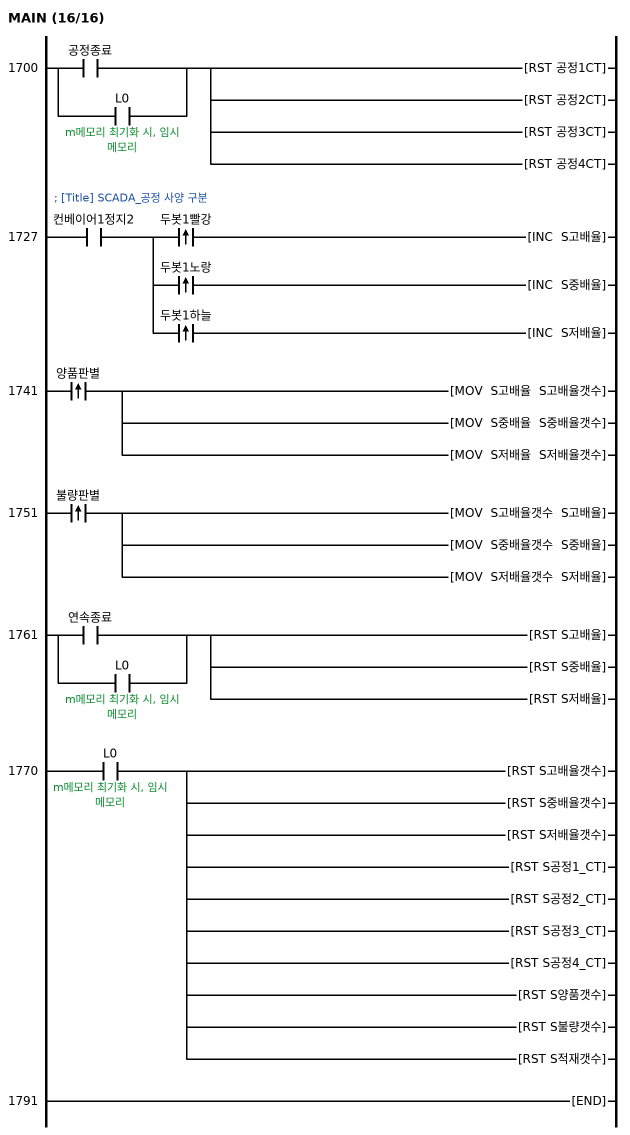
1700  LD      공정종료
      OR      L0  ; m메모리 최기화 시, 임시 메모리
      RST     공정1CT
      RST     공정2CT
      RST     공정3CT
      RST     공정4CT
; [Title] SCADA_공정 사양 구분
1727  LD      컨베이어1정지2
      MPS
      ANDP    두봇1빨강
      INC     S고배율
      MRD
      ANDP    두봇1노랑
      INC     S중배율
      MPP
      ANDP    두봇1하늘
      INC     S저배율
1741  LDP     양품판별
      MOV     S고배율 S고배율갯수
      MOV     S중배율 S중배율갯수
      MOV     S저배율 S저배율갯수
1751  LDP     불량판별
      MOV     S고배율갯수 S고배율
      MOV     S중배율갯수 S중배율
      MOV     S저배율갯수 S저배율
1761  LD      연속종료
      OR      L0  ; m메모리 최기화 시, 임시 메모리
      RST     S고배율
      RST     S중배율
      RST     S저배율
1770  LD      L0  ; m메모리 최기화 시, 임시 메모리
      RST     S고배율갯수
      RST     S중배율갯수
      RST     S저배율갯수
      RST     S공정1_CT
      RST     S공정2_CT
      RST     S공정3_CT
      RST     S공정4_CT
      RST     S양품갯수
      RST     S불량갯수
      RST     S적재갯수
1791  END
END_PROGRAM

// device comments not shown above
Y44  ; 1축서보정지
Y45  ; 2축서보정지
D0  ; n번쨰공정
D10  ; 공급주문갯수
D30  ; 물건지나간갯수
D40  ; H전압값
M23  ; '
M90  ; 비상정지셋
M767  ; H공급전진
M768  ; H공급후진
M769  ; H셀정지전진
M770  ; H셀정지후진
M771  ; H전극정지전진
M772  ; H전극정지후진
M773  ; H전극측정실린더
M774  ; H뚜껑압착전진
M775  ; H뚜껑압착후진
M776  ; H케이스장착실린더
M777  ; H적재전진
M778  ; H적재후진
M874  ; 주문갯수틀렸을시공급중단
M990  ; 서보위치결정완료신호1
M991  ; 서보위치결정완료2
M992  ; 서보위치결정완료3
M993  ; 서보위치결정완료4
M994  ; 서보위치결정완료5
M995  ; 서보위치결정완료6
M996  ; 서보위치결정완료7
M997  ; 서보위치결정완료4
M998  ; 서보위치결정완료신호3
M999  ; 서보위치결정완료신호2
M1102  ; 모든공정종료신호
M2500  ; ]
D45  ; H무게값
D203  ; 실제공급한갯수
D350  ; 1축조그속도표시
D370  ; 2축조그속도표시
D874  ; 공급
T0  ; 전압정지타이머
T1  ; 전압측정솔타이머
T2  ; 비전검수대기타이머
T3  ; 모터역,정 회전타이밍
T4  ; 케이스장착대기타이머
T5  ; 케이스장착대기타이머2
T6  ; 모터회전딜레이타이머
T7  ; 모터회전대기타이머2
T8  ; 케이스압착공정타이머
